// TIA Portal V20 export
FUNCTION_BLOCK "LER_WeightCheck"   // FB121, LAD
// stored: Access Published, MemoryReserve 100, SetENOAutomatically false
   VAR_INPUT
      enable : Bool;
      enableManualCmds : Bool;
      dryRunCmds : Bool;
      simulationCmds : Bool;
   END_VAR
   VAR_OUTPUT
      error : Bool;
      errorCode : Word;
   END_VAR
   VAR_IN_OUT
      configuration : "LER_WeightCheckConfiguration";
      moduleInterface : "LER_WeightCheckInterface";
      controlNode : "LER_WeightCheckControlNode";
   END_VAR
   VAR
      instTON_completeDelay : TON_TIME;
      instTON_system : Array[0..1] of TON_TIME;
      instTON_scale : Array[0..1] of TON_TIME;
      statTonTimer { S7_SetPoint := 'True'} : Array[0..99] of TON_TIME;
      statMonitoring : "LER_WeightCheckMonitoring";
      statRetValInt : Array[1..#count] of Int;
      statRetValWord : Array[1..#count] of Word;
      statPulse : Array[0..99] of Bool;
      statByteToBool : Struct
         zeroSetCmd : Bool;
         calibrationCmd : Bool;
         ambientConditionCmd : Bool;
         systemAlive : Bool;
         scaleAlive : Bool;
         zeroSetBusy : Bool;
         calibrationBusy : Bool;
         ambientConditionBusy : Bool;
         zeroSetCompletion : Bool;
         calibrationCompletion : Bool;
         ambientConditionCompletion : Bool;
         zeroSetError : Bool;
         calibrationError : Bool;
         ambientConditionError : Bool;
         calibrationStatusBusy : Bool;
         calibrationStatusIdle : Bool;
         calibrationStatusDetect : Bool;
         calibrationStatusCompletion : Bool;
         calibrationStatusError : Bool;
         stable : Bool;
      END_STRUCT;
      statHeartBit_system : Bool;
      statHeartBit_scale : Bool;
      statRowDataDword_capture : DWord;
      statRowDataReal_capture : Real;
      statRowDataDint_capture : DInt;
      statRowDataDword_always : DWord;
      statRowDataReal_always : Real;
      statRowDataDint_always : DInt;
   END_VAR
   VAR_TEMP
      tempRetVal : Array[1..#count] of Int;
      tempIndex : Int;
   END_VAR
   VAR CONSTANT
      delayTime : Time := T#3s;
      count : Int := 5;
      statusNoErrorOccurred : Word := 16#0000;   // No error occurred.
      errHeartBit : Word := 16#8000;
      errScaleStatus : Word := 16#8001;
      errHwdNotConfigured : Word := 16#8090;   // You have not configured a module for the specified hardware identifier or You have ignored the restriction concerning the length of consistent data, or you have not specified a hardware identifier as an address at parameter LADDR
      errRecordDataType : Word := 16#8092;   // Non-supported data type in the RECORD parameter.
      errNoDpProfinetIoModule : Word := 16#8093;   // No DP module/PROFINET IO device from which you can read consistent data exists for the hardware identifier specified in LADDR . This error code also occurs if the module addressed by means of LADDR does not have inputs.
      errIoAccessPermission : Word := 16#80A0;   // An access error was detected when accessing the I/O.
      errRecordLengthInsufficient : Word := 16#80B1;   // The length of the specified destination area at parameter RECORD is shorter than the configured user data length.
      errDataNotReceived : Word := 16#80C0;   // The data have not been read yet.
   END_VAR
   VAR_TEMP   // added for the SCL form of the ladder/FBD networks
      _w1 : Bool;
      _w2 : Bool;
      _w3 : Bool;
      _w4 : Bool;
   END_VAR
BEGIN

REGION Network 1 (SCL): DP READ
   REGION DP read

       IF #enable AND NOT #simulationCmds THEN
           #"statRetValInt"[1] := DPRD_DAT(LADDR := #configuration.hwID.pncMainStatusID, RECORD => #statMonitoring.profinetInput.pncMainStatus);
           #"statRetValInt"[2] := DPRD_DAT(LADDR := #configuration.hwID.scaleStatusID, RECORD => #statMonitoring.profinetInput.scaleStatus);
       END_IF;

   END_REGION
END_REGION

REGION Network 2 (SCL): INPUT MAPPING
   REGION Input mapping

       // pncMainStatus
       #statByteToBool.systemAlive := #statMonitoring.profinetInput.pncMainStatus.systemAlive.%X0;

       // scaleStatus
       #statByteToBool.scaleAlive := #statMonitoring.profinetInput.scaleStatus.scaleAlive.%X0;

       #statByteToBool.zeroSetBusy := #statMonitoring.profinetInput.scaleStatus.cmdResponse.%X0;
       #statByteToBool.calibrationBusy := #statMonitoring.profinetInput.scaleStatus.cmdResponse.%X1;
       #statByteToBool.ambientConditionBusy := #statMonitoring.profinetInput.scaleStatus.cmdResponse.%X2;

       #statByteToBool.zeroSetCompletion := #statMonitoring.profinetInput.scaleStatus.cmdCompletion.%X0;
       #statByteToBool.calibrationCompletion := #statMonitoring.profinetInput.scaleStatus.cmdCompletion.%X1;
       #statByteToBool.ambientConditionCompletion := #statMonitoring.profinetInput.scaleStatus.cmdCompletion.%X2;

       #statByteToBool.zeroSetError := #statMonitoring.profinetInput.scaleStatus.cmdError.%X0;
       #statByteToBool.calibrationError := #statMonitoring.profinetInput.scaleStatus.cmdError.%X1;
       #statByteToBool.ambientConditionError := #statMonitoring.profinetInput.scaleStatus.cmdError.%X2;

       #statByteToBool.calibrationStatusBusy := NOT #statMonitoring.profinetInput.scaleStatus.calibrationStatus.%X0;
       #statByteToBool.calibrationStatusIdle := #statMonitoring.profinetInput.scaleStatus.calibrationStatus.%X0;
       #statByteToBool.calibrationStatusDetect := #statMonitoring.profinetInput.scaleStatus.calibrationStatus.%X1;
       #statByteToBool.calibrationStatusCompletion := #statMonitoring.profinetInput.scaleStatus.calibrationStatus.%X0 OR #statMonitoring.profinetInput.scaleStatus.calibrationStatus.%X1;
       #statByteToBool.calibrationStatusError := #statMonitoring.profinetInput.scaleStatus.calibrationStatus.%X7;

       #statByteToBool.stable := #statMonitoring.profinetInput.scaleStatus.stableStatus.%X0;

           // Parameter setting SV move 
       IF #controlNode.command.configSave THEN
           #moduleInterface.monitoring.weightRangeMinPV := #moduleInterface.configuration.weightRangeMinSV;
           #moduleInterface.monitoring.weightRangeMaxPV := #moduleInterface.configuration.weightRangeMaxSV;
       END_IF;

   END_REGION
END_REGION

REGION Network 3 (SCL): ERROR STATUS
   REGION Error check

       IF #enable AND NOT #simulationCmds THEN
           IF #statByteToBool.zeroSetError OR
               #statByteToBool.calibrationError OR
               #statByteToBool.ambientConditionError OR
               #statByteToBool.calibrationStatusError THEN
               #errorCode := #errScaleStatus;

           ELSIF #statRetValInt <> #tempRetVal THEN
               FOR #tempIndex := 1 TO #count DO
                   #statRetValWord[#tempIndex] := INT_TO_WORD(#statRetValInt[#tempIndex]);
                   CASE #statRetValWord[#tempIndex] OF

                       #errHwdNotConfigured:
                           #errorCode := #errHwdNotConfigured;

                       #errRecordDataType:
                           #errorCode := #errRecordDataType;

                       #errNoDpProfinetIoModule:
                           #errorCode := #errNoDpProfinetIoModule;

                       #errIoAccessPermission:
                           #errorCode := #errIoAccessPermission;

                       #errRecordLengthInsufficient:
                           #errorCode := #errRecordLengthInsufficient;

                       #errDataNotReceived:
                           #errorCode := #errDataNotReceived;
                   END_CASE;
               END_FOR;
           ELSE
               #errorCode := #statusNoErrorOccurred;
           END_IF;
       ELSE
           #errorCode := #statusNoErrorOccurred;
       END_IF;

       #error := #errorCode <> 0;
       #statMonitoring.error := #error;

   END_REGION
END_REGION

REGION Network 4: SEQUENCE : READY
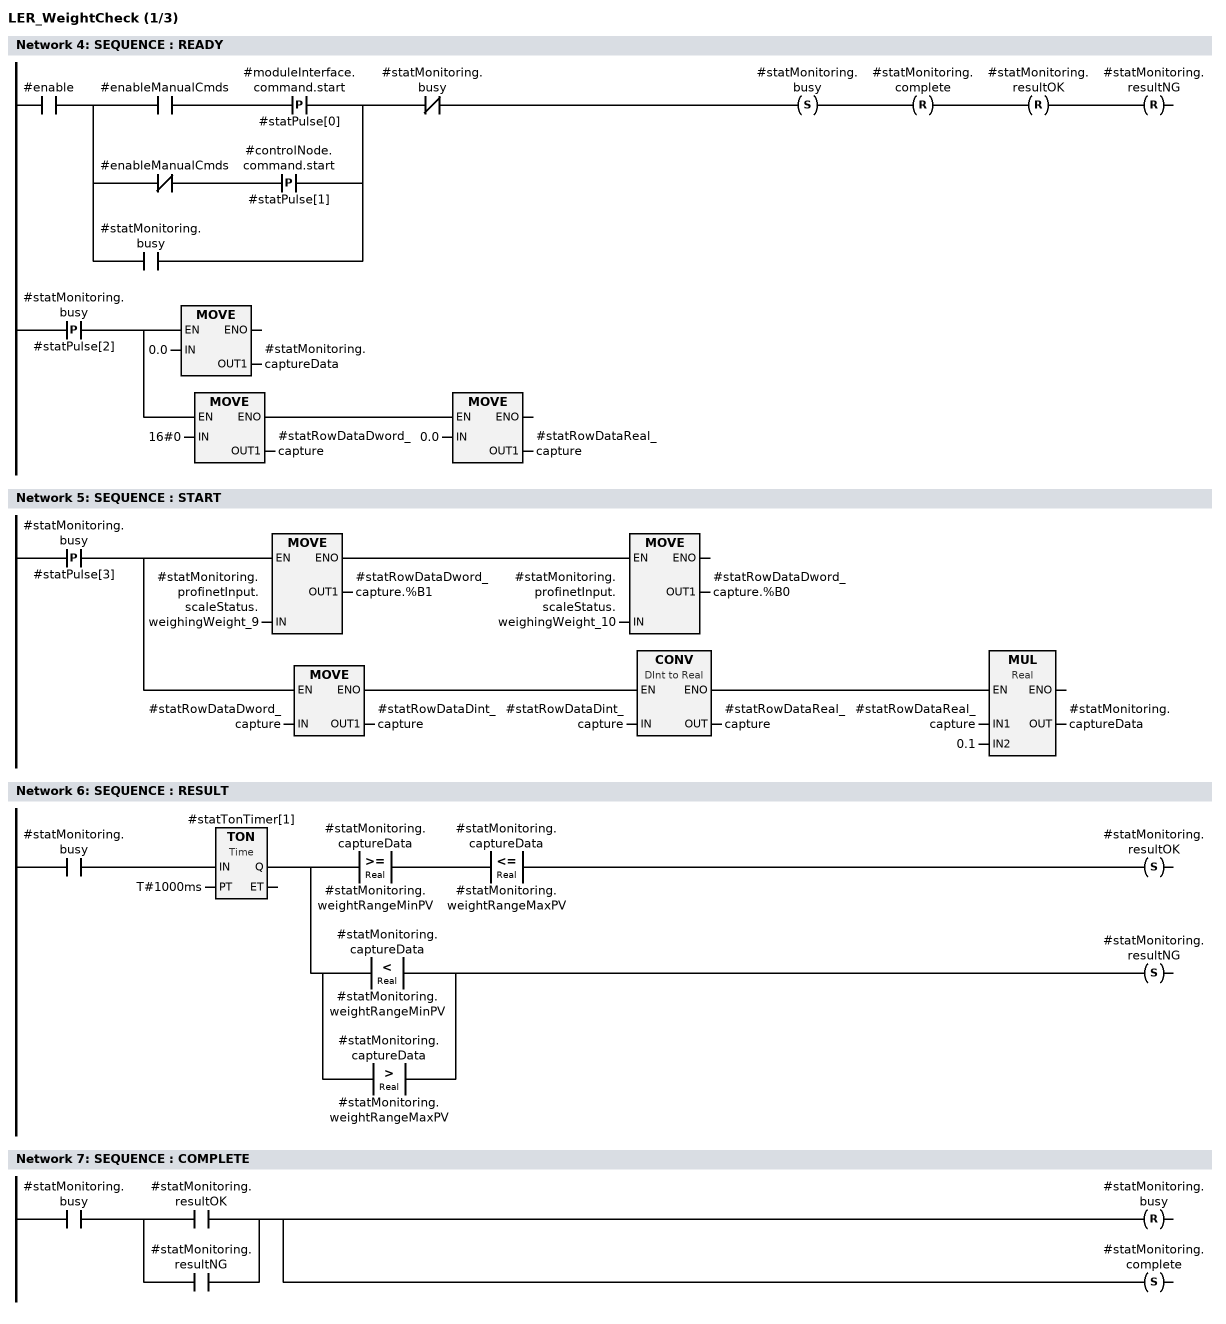
   RUNG wire#powerrail
      Contact( #enable )
      wire#w1
      Contact( #enableManualCmds )
      P_Contact(operand := #moduleInterface.command.start, bit := #statPulse[0])
      wire#w2
      I_Contact( #statMonitoring.busy )
      S_Coil( #statMonitoring.busy )
      R_Coil( #statMonitoring.complete )
      R_Coil( #statMonitoring.resultOK )
      R_Coil( #statMonitoring.resultNG )
   END_RUNG
   RUNG wire#w1
      I_Contact( #enableManualCmds )
      P_Contact(operand := #controlNode.command.start, bit := #statPulse[1])
   END_RUNG wire#w2
   RUNG wire#w1
      Contact( #statMonitoring.busy )
   END_RUNG wire#w2
   RUNG wire#powerrail
      P_Contact(operand := #statMonitoring.busy, bit := #statPulse[2])
      wire#w3
      Move(in := 0.0, out1 => #statMonitoring.captureData)
   END_RUNG
   RUNG wire#w3
      Move(in := 16#0, out1 => #statRowDataDword_capture)
      Move(in := 0.0, out1 => #statRowDataReal_capture)
   END_RUNG
   // the same network as SCL:
   #_w1 := #enable AND #enableManualCmds AND #moduleInterface.command.start AND NOT #statPulse[0];   // rising edge of #moduleInterface.command.start
   #statPulse[0] := #moduleInterface.command.start;
   #_w2 := #enable AND NOT #enableManualCmds AND #controlNode.command.start AND NOT #statPulse[1];   // rising edge of #controlNode.command.start
   #statPulse[1] := #controlNode.command.start;
   #_w3 := (#_w1 OR #_w2 OR (#enable AND #statMonitoring.busy)) AND NOT #statMonitoring.busy;
   IF #_w3 THEN
       #statMonitoring.busy := TRUE;
       #statMonitoring.complete := FALSE;
       #statMonitoring.resultOK := FALSE;
       #statMonitoring.resultNG := FALSE;
   END_IF;
   #_w4 := #statMonitoring.busy AND NOT #statPulse[2];   // rising edge of #statMonitoring.busy
   #statPulse[2] := #statMonitoring.busy;
   IF #_w4 THEN
       #statMonitoring.captureData := 0.0;
       #statRowDataDword_capture := 16#0;
       #statRowDataReal_capture := 0.0;
   END_IF;
END_REGION

REGION Network 5: SEQUENCE : START
   RUNG wire#powerrail
      P_Contact(operand := #statMonitoring.busy, bit := #statPulse[3])
      wire#w1
      Move(in := #statMonitoring.profinetInput.scaleStatus.weighingWeight_9, out1 => #statRowDataDword_capture.%B1)
      Move(in := #statMonitoring.profinetInput.scaleStatus.weighingWeight_10, out1 => #statRowDataDword_capture.%B0)
   END_RUNG
   RUNG wire#w1
      Move(in := #statRowDataDword_capture, out1 => #statRowDataDint_capture)
      { S7_Templates := "[SrcType := DInt, DestType := Real]" } Convert(in := #statRowDataDint_capture, out => #statRowDataReal_capture)
      { S7_Templates := "SrcType := Real" } Mul(in1 := #statRowDataReal_capture, in2 := 0.1, out => #statMonitoring.captureData)
   END_RUNG
   // the same network as SCL:
   #_w1 := #statMonitoring.busy AND NOT #statPulse[3];   // rising edge of #statMonitoring.busy
   #statPulse[3] := #statMonitoring.busy;
   IF #_w1 THEN
       #statRowDataDword_capture.%B1 := #statMonitoring.profinetInput.scaleStatus.weighingWeight_9;
       #statRowDataDword_capture.%B0 := #statMonitoring.profinetInput.scaleStatus.weighingWeight_10;
       #statRowDataDint_capture := #statRowDataDword_capture;
       #statRowDataReal_capture := DINT_TO_REAL(#statRowDataDint_capture);
       #statMonitoring.captureData := #statRowDataReal_capture * 0.1;
   END_IF;
END_REGION

REGION Network 6: SEQUENCE : RESULT
   RUNG wire#powerrail
      Contact( #statMonitoring.busy )
      { S7_Templates := "time_type := Time" } #statTonTimer[1].TON(pt := T#1000ms, et =>)
      wire#w1
      { S7_Templates := "SrcType := Real" } GE_Contact(in1 := #statMonitoring.captureData, in2 := #statMonitoring.weightRangeMinPV)
      { S7_Templates := "SrcType := Real" } LE_Contact(in1 := #statMonitoring.captureData, in2 := #statMonitoring.weightRangeMaxPV)
      S_Coil( #statMonitoring.resultOK )
   END_RUNG
   RUNG wire#w1
      { S7_Templates := "SrcType := Real" } LT_Contact(in1 := #statMonitoring.captureData, in2 := #statMonitoring.weightRangeMinPV)
      wire#w2
      S_Coil( #statMonitoring.resultNG )
   END_RUNG
   RUNG wire#w1
      { S7_Templates := "SrcType := Real" } GT_Contact(in1 := #statMonitoring.captureData, in2 := #statMonitoring.weightRangeMaxPV)
   END_RUNG wire#w2
   // the same network as SCL:
   #statTonTimer[1].TON(IN := #statMonitoring.busy, PT := T#1000ms);
   IF #statTonTimer[1].Q AND (#statMonitoring.captureData >= #statMonitoring.weightRangeMinPV) AND (#statMonitoring.captureData <= #statMonitoring.weightRangeMaxPV) THEN
       #statMonitoring.resultOK := TRUE;
   END_IF;
   IF #statTonTimer[1].Q AND ((#statMonitoring.captureData < #statMonitoring.weightRangeMinPV) OR (#statMonitoring.captureData > #statMonitoring.weightRangeMaxPV)) THEN
       #statMonitoring.resultNG := TRUE;
   END_IF;
END_REGION

REGION Network 7: SEQUENCE : COMPLETE
   RUNG wire#powerrail
      Contact( #statMonitoring.busy )
      wire#w1
      Contact( #statMonitoring.resultOK )
      wire#w2
      R_Coil( #statMonitoring.busy )
   END_RUNG
   RUNG wire#w1
      Contact( #statMonitoring.resultNG )
   END_RUNG wire#w2
   RUNG wire#w2
      S_Coil( #statMonitoring.complete )
   END_RUNG
   // the same network as SCL:
   #_w1 := #statMonitoring.busy AND (#statMonitoring.resultOK OR #statMonitoring.resultNG);
   IF #_w1 THEN
       #statMonitoring.busy := FALSE;
       #statMonitoring.complete := TRUE;
   END_IF;
END_REGION

REGION Network 8: ALWAYS DATA SAVE
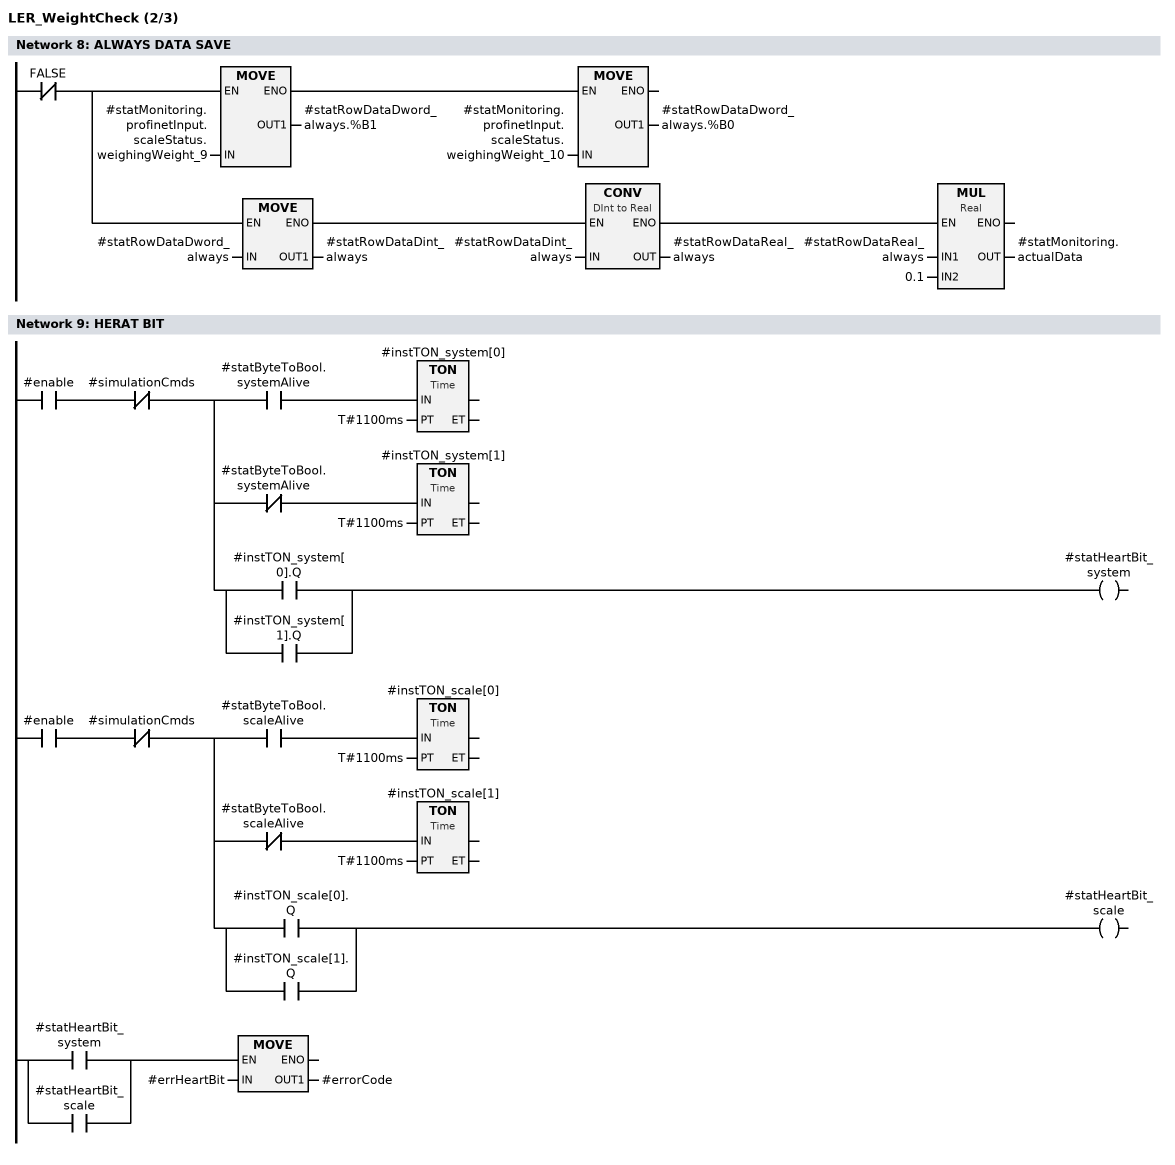
   RUNG wire#powerrail
      I_Contact( FALSE )
      wire#w1
      Move(in := #statMonitoring.profinetInput.scaleStatus.weighingWeight_9, out1 => #statRowDataDword_always.%B1)
      Move(in := #statMonitoring.profinetInput.scaleStatus.weighingWeight_10, out1 => #statRowDataDword_always.%B0)
   END_RUNG
   RUNG wire#w1
      Move(in := #statRowDataDword_always, out1 => #statRowDataDint_always)
      { S7_Templates := "[SrcType := DInt, DestType := Real]" } Convert(in := #statRowDataDint_always, out => #statRowDataReal_always)
      { S7_Templates := "SrcType := Real" } Mul(in1 := #statRowDataReal_always, in2 := 0.1, out => #statMonitoring.actualData)
   END_RUNG
   // the same network as SCL:
   IF NOT FALSE THEN
       #statRowDataDword_always.%B1 := #statMonitoring.profinetInput.scaleStatus.weighingWeight_9;
       #statRowDataDword_always.%B0 := #statMonitoring.profinetInput.scaleStatus.weighingWeight_10;
       #statRowDataDint_always := #statRowDataDword_always;
       #statRowDataReal_always := DINT_TO_REAL(#statRowDataDint_always);
       #statMonitoring.actualData := #statRowDataReal_always * 0.1;
   END_IF;
END_REGION

REGION Network 9: HERAT BIT
   RUNG wire#powerrail
      Contact( #enable )
      I_Contact( #simulationCmds )
      wire#w1
      Contact( #statByteToBool.systemAlive )
      { S7_Templates := "time_type := Time" } #instTON_system[0].TON(pt := T#1100ms, et =>)
   END_RUNG
   RUNG wire#w1
      I_Contact( #statByteToBool.systemAlive )
      { S7_Templates := "time_type := Time" } #instTON_system[1].TON(pt := T#1100ms, et =>)
   END_RUNG
   RUNG wire#w1
      Contact( #instTON_system[0].Q )
      wire#w2
      Coil( #statHeartBit_system )
   END_RUNG
   RUNG wire#w1
      Contact( #instTON_system[1].Q )
   END_RUNG wire#w2
   RUNG wire#powerrail
      Contact( #enable )
      I_Contact( #simulationCmds )
      wire#w3
      Contact( #statByteToBool.scaleAlive )
      { S7_Templates := "time_type := Time" } #instTON_scale[0].TON(pt := T#1100ms, et =>)
   END_RUNG
   RUNG wire#w3
      I_Contact( #statByteToBool.scaleAlive )
      { S7_Templates := "time_type := Time" } #instTON_scale[1].TON(pt := T#1100ms, et =>)
   END_RUNG
   RUNG wire#w3
      Contact( #instTON_scale[0].Q )
      wire#w4
      Coil( #statHeartBit_scale )
   END_RUNG
   RUNG wire#w3
      Contact( #instTON_scale[1].Q )
   END_RUNG wire#w4
   RUNG wire#powerrail
      Contact( #statHeartBit_system )
      wire#w5
      Move(in := #errHeartBit, out1 => #errorCode)
   END_RUNG
   RUNG wire#powerrail
      Contact( #statHeartBit_scale )
   END_RUNG wire#w5
   // the same network as SCL:
   #_w1 := #enable AND NOT #simulationCmds;
   #instTON_system[0].TON(IN := #_w1 AND #statByteToBool.systemAlive, PT := T#1100ms);
   #instTON_system[1].TON(IN := #_w1 AND NOT #statByteToBool.systemAlive, PT := T#1100ms);
   #statHeartBit_system := #_w1 AND (#instTON_system[0].Q OR #instTON_system[1].Q);
   #_w2 := #enable AND NOT #simulationCmds;
   #instTON_scale[0].TON(IN := #_w2 AND #statByteToBool.scaleAlive, PT := T#1100ms);
   #instTON_scale[1].TON(IN := #_w2 AND NOT #statByteToBool.scaleAlive, PT := T#1100ms);
   #statHeartBit_scale := #_w2 AND (#instTON_scale[0].Q OR #instTON_scale[1].Q);
   IF #statHeartBit_system OR #statHeartBit_scale THEN #errorCode := #errHeartBit; END_IF;
END_REGION

REGION Network 10: CONFIGURATION
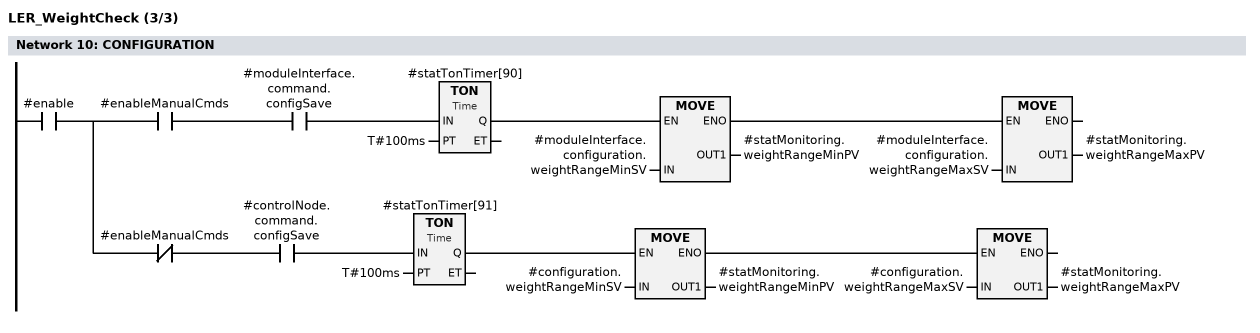
   RUNG wire#powerrail
      Contact( #enable )
      wire#w1
      Contact( #enableManualCmds )
      Contact( #moduleInterface.command.configSave )
      { S7_Templates := "time_type := Time" } #statTonTimer[90].TON(pt := T#100ms, et =>)
      Move(in := #moduleInterface.configuration.weightRangeMinSV, out1 => #statMonitoring.weightRangeMinPV)
      Move(in := #moduleInterface.configuration.weightRangeMaxSV, out1 => #statMonitoring.weightRangeMaxPV)
   END_RUNG
   RUNG wire#w1
      I_Contact( #enableManualCmds )
      Contact( #controlNode.command.configSave )
      { S7_Templates := "time_type := Time" } #statTonTimer[91].TON(pt := T#100ms, et =>)
      Move(in := #configuration.weightRangeMinSV, out1 => #statMonitoring.weightRangeMinPV)
      Move(in := #configuration.weightRangeMaxSV, out1 => #statMonitoring.weightRangeMaxPV)
   END_RUNG
   // the same network as SCL:
   #statTonTimer[90].TON(IN := #enable AND #enableManualCmds AND #moduleInterface.command.configSave,
                         PT := T#100ms);
   IF #statTonTimer[90].Q THEN
       #statMonitoring.weightRangeMinPV := #moduleInterface.configuration.weightRangeMinSV;
       #statMonitoring.weightRangeMaxPV := #moduleInterface.configuration.weightRangeMaxSV;
   END_IF;
   #statTonTimer[91].TON(IN := #enable AND NOT #enableManualCmds AND #controlNode.command.configSave,
                         PT := T#100ms);
   IF #statTonTimer[91].Q THEN
       #statMonitoring.weightRangeMinPV := #configuration.weightRangeMinSV;
       #statMonitoring.weightRangeMaxPV := #configuration.weightRangeMaxSV;
   END_IF;
END_REGION

REGION Network 11 (SCL): DP WRITE
   REGION DP write

       IF #enable AND NOT #simulationCmds THEN
           #"statRetValInt"[3] := DPWR_DAT(LADDR := #configuration.hwID.scaleControlID, RECORD := #statMonitoring.profinetOutput.scaleControl);
       END_IF;

   END_REGION
END_REGION

REGION Network 12 (SCL): OUTPUT MAPPING
   REGION Output mapping

       IF #enable THEN
           //pncCmd
           #statMonitoring.profinetOutput.scaleControl.pncCmd.%X0 := #statByteToBool.zeroSetCmd; // Zero set is adjusting the offset(simple adjustment).
           #statMonitoring.profinetOutput.scaleControl.pncCmd.%X1 := #statByteToBool.calibrationCmd; // Calibration is adjusting the scale(details adjustment).
           #statMonitoring.profinetOutput.scaleControl.pncCmd.%X2 := #statByteToBool.ambientConditionCmd;

           #controlNode.monitoring := #moduleInterface.monitoring := #statMonitoring;
       END_IF;

   END_REGION
END_REGION
END_FUNCTION_BLOCK
